TEXTLIST EL2809_M_3
  1 = 'Vac Pump Run/Stop' | chinese: '真空吸附启停' | Chinese: '真空吸附启停'
  2 = 'Cylinder S2 rises' | chinese: '压辊气缸S2上升' | Chinese: '压辊气缸S2上升'
  3 = 'Cylinder S3 rises' | chinese: '压辊气缸S3上升' | Chinese: '压辊气缸S3上升'
  4 = 'Cylinder S4 rises' | chinese: '压辊气缸S4上升' | Chinese: '压辊气缸S4上升'
  5 = 'Cylinder S5 rises' | chinese: '压辊气缸S5上升' | Chinese: '压辊气缸S5上升'
  6 = 'Cylinder S6 rises' | chinese: '压辊气缸S6上升' | Chinese: '压辊气缸S6上升'
  7 = 'Cylinder S2 drops' | chinese: '压辊气缸S2下降' | Chinese: '压辊气缸S2下降'
  8 = 'Cylinder S3 drops' | chinese: '压辊气缸S3下降' | Chinese: '压辊气缸S3下降'
  9 = 'Cylinder S4 drops' | chinese: '压辊气缸S4下降' | Chinese: '压辊气缸S4下降'
  10 = 'Cylinder S5 drops' | chinese: '压辊气缸S5下降' | Chinese: '压辊气缸S5下降'
  11 = 'Cylinder S6 drops' | chinese: '压辊气缸S6下降' | Chinese: '压辊气缸S6下降'
  12 = ''
  13 = ''
  14 = ''
  15 = ''
  16 = ''
   = ''
END_TEXTLIST

(* stored: Version 1.1.0.1, ProductVersion 3.1.4024.11
   TextList EL2809_M_3: Id {15e7d1ac-6127-4b1c-8184-53ae704069ad} *)
